# EPICS substitutions: ngpspsuSup/status_hex.substitutions
file status_hex.template {

pattern {P, INDEX}
{"\$(P)", "1"}
{"\$(P)", "2"}
{"\$(P)", "3"}
{"\$(P)", "4"}
{"\$(P)", "5"}
{"\$(P)", "6"}
{"\$(P)", "7"}
{"\$(P)", "8"}
}
